PROGRAM MAIN
VAR
    // This is the single instance of our entire modular machine.
    // By keeping it here, we keep the global namespace perfectly clean.
	{attribute 'OPC.UA.DA' := '1'}
    RotaryCutter : FB_MainMachine;
END_VAR

// =========================================================
// 1. HARDWARE / SIMULATION MULTIPLEXER
// =========================================================
IF GVL_Safety.bSimulationMode THEN
    GVL_Safety.bSafetyOk := GVL_Safety.bSimulateSafety;
ELSE
    GVL_Safety.bSafetyOk := GVL_Safety.bPhysicalSafetyOk;
END_IF

// =========================================================
// 2. EXECUTE THE MACHINE
// =========================================================
RotaryCutter();

END_PROGRAM

(* stored: Version 1.1.0.1
   POU MAIN: Id {4d0baa44-d475-46c3-a965-e7a9bb8474bf}, SpecialFunc None *)
